	PROC longwelds()
		MoveJ [[-537.74,1528.93,225.26],[0.133056,-0.223334,0.96556,0.0105691],[1,-1,1,0],[9E+09,9E+09,9E+09,9E+09,9E+09,9E+09]], v1000, z50, tWeldGun;
		MoveJ [[-534.17,1676.79,-7.31],[0.13306,-0.223351,0.965556,0.0105536],[1,-1,1,0],[9E+09,9E+09,9E+09,9E+09,9E+09,9E+09]], v1000, z50, tWeldGun;
		ArcLStart [[-534.18,1676.79,-10.95],[0.13306,-0.223361,0.965554,0.0105477],[1,-1,1,0],[9E+09,9E+09,9E+09,9E+09,9E+09,9E+09]], v30, seam13, weld13, fine, tWeldGun;
		ArcL [[-544.58,1676.80,-10.94],[0.133063,-0.223367,0.965552,0.0105509],[1,-1,1,0],[9E+09,9E+09,9E+09,9E+09,9E+09,9E+09]], v30, seam13, weld13, z10, tWeldGun;
		ArcL [[-560.58,1676.80,-10.94],[0.133064,-0.223373,0.96555,0.0105523],[1,-1,1,0],[9E+09,9E+09,9E+09,9E+09,9E+09,9E+09]], v30, seam13, weld13, z10, tWeldGun;
		ArcLEnd [[-573.39,1676.78,-10.94],[0.133047,-0.223358,0.965556,0.0105449],[1,-1,1,0],[9E+09,9E+09,9E+09,9E+09,9E+09,9E+09]], v30, seam13, weld13, fine, tWeldGun;
		MoveL [[-573.40,1676.83,-5.98],[0.133038,-0.223382,0.965552,0.0105696],[1,-1,1,0],[9E+09,9E+09,9E+09,9E+09,9E+09,9E+09]], v50, z1, tWeldGun;
		MoveL [[-575.35,1723.62,-6.01],[0.133042,-0.223378,0.965552,0.0105594],[1,-1,1,0],[9E+09,9E+09,9E+09,9E+09,9E+09,9E+09]], v50, z1, tWeldGun;
		ArcLStart [[-575.34,1723.62,-15.03],[0.133047,-0.22338,0.965551,0.0105632],[1,-1,1,0],[9E+09,9E+09,9E+09,9E+09,9E+09,9E+09]], v30, seam13, weld13, fine, tWeldGun;
		ArcL [[-575.34,1697.62,-15.03],[0.133047,-0.22338,0.965551,0.0105669],[1,-1,1,0],[9E+09,9E+09,9E+09,9E+09,9E+09,9E+09]], v30, seam13, weld13, fine, tWeldGun;
		ArcL [[-575.35,1676.62,-15.02],[0.133043,-0.223381,0.965552,0.0105654],[1,-1,1,0],[9E+09,9E+09,9E+09,9E+09,9E+09,9E+09]], v30, seam13, weld13, fine, tWeldGun;
		ArcL [[-575.35,1655.62,-15.02],[0.13304,-0.223383,0.965551,0.010569],[1,-1,1,0],[9E+09,9E+09,9E+09,9E+09,9E+09,9E+09]], v30, seam13, weld13, fine, tWeldGun;
		ArcL [[-575.35,1632.62,-15.03],[0.133037,-0.22338,0.965553,0.0105659],[1,-1,1,0],[9E+09,9E+09,9E+09,9E+09,9E+09,9E+09]], v30, seam13, weld13, fine, tWeldGun;
		ArcLEnd [[-575.35,1606.61,-15.03],[0.133037,-0.223381,0.965552,0.0105613],[1,-1,1,0],[9E+09,9E+09,9E+09,9E+09,9E+09,9E+09]], v30, seam13, weld13, fine, tWeldGun;
		MoveL [[-575.35,1606.60,-1.09],[0.13303,-0.223389,0.965551,0.0105647],[1,-1,1,0],[9E+09,9E+09,9E+09,9E+09,9E+09,9E+09]], v50, z1, tWeldGun;
		MoveL [[-575.34,1585.59,-1.13],[0.133025,-0.223396,0.965551,0.0105485],[1,-1,1,0],[9E+09,9E+09,9E+09,9E+09,9E+09,9E+09]], v50, z1, tWeldGun;
		ArcLStart [[-574.36,1584.60,-16.12],[0.133023,-0.223401,0.96555,0.010553],[1,-1,1,0],[9E+09,9E+09,9E+09,9E+09,9E+09,9E+09]], v30, seam13, weld13\Weave:=weave1, fine, tWeldGun;
		ArcL [[-574.36,1575.59,-16.13],[0.13302,-0.2234,0.96555,0.0105496],[1,-1,1,0],[9E+09,9E+09,9E+09,9E+09,9E+09,9E+09]], v30, seam13, weld13\Weave:=weave1, fine, tWeldGun;
		ArcL [[-573.36,1542.60,-16.12],[0.133024,-0.223405,0.965549,0.0105554],[1,-1,1,0],[9E+09,9E+09,9E+09,9E+09,9E+09,9E+09]], v30, seam13, weld13\Weave:=weave1, fine, tWeldGun;
		ArcL [[-573.37,1523.59,-16.12],[0.133018,-0.223399,0.965551,0.010556],[1,-1,1,0],[9E+09,9E+09,9E+09,9E+09,9E+09,9E+09]], v30, seam13, weld13\Weave:=weave1, fine, tWeldGun;
		ArcLEnd [[-573.36,1500.60,-16.12],[0.133023,-0.223402,0.965549,0.0105616],[1,-1,1,0],[9E+09,9E+09,9E+09,9E+09,9E+09,9E+09]], v30, seam13, weld13\Weave:=weave1, fine, tWeldGun;
		MoveL [[-573.39,1500.62,-2.23],[0.132981,-0.22343,0.965549,0.0105695],[1,-1,1,0],[9E+09,9E+09,9E+09,9E+09,9E+09,9E+09]], v50, z1, tWeldGun;
		MoveL [[-573.39,1485.63,-2.25],[0.132987,-0.223446,0.965544,0.0105683],[1,-1,1,0],[9E+09,9E+09,9E+09,9E+09,9E+09,9E+09]], v50, z1, tWeldGun;
		ArcLStart [[-573.39,1485.63,-15.25],[0.132986,-0.223448,0.965544,0.0105658],[1,-1,1,0],[9E+09,9E+09,9E+09,9E+09,9E+09,9E+09]], v30, seam13, weld13\Weave:=weave1, fine, tWeldGun;
		ArcL [[-573.40,1464.62,-15.25],[0.132977,-0.223444,0.965546,0.0105643],[1,-1,1,0],[9E+09,9E+09,9E+09,9E+09,9E+09,9E+09]], v30, seam13, weld13\Weave:=weave1, fine, tWeldGun;
		ArcL [[-574.40,1445.63,-15.24],[0.132983,-0.223455,0.965542,0.0105677],[1,-1,1,0],[9E+09,9E+09,9E+09,9E+09,9E+09,9E+09]], v30, seam13, weld13\Weave:=weave1, fine, tWeldGun;
		ArcL [[-574.40,1425.64,-15.24],[0.132985,-0.223457,0.965542,0.0105723],[1,-1,1,0],[9E+09,9E+09,9E+09,9E+09,9E+09,9E+09]], v30, seam13, weld13\Weave:=weave1, fine, tWeldGun;
		ArcL [[-574.40,1404.65,-15.23],[0.132998,-0.223476,0.965536,0.0105691],[1,-1,1,0],[9E+09,9E+09,9E+09,9E+09,9E+09,9E+09]], v30, seam13, weld13\Weave:=weave1, fine, tWeldGun;
		ArcL [[-574.41,1387.63,-15.25],[0.132976,-0.223459,0.965543,0.0105667],[1,-1,1,0],[9E+09,9E+09,9E+09,9E+09,9E+09,9E+09]], v30, seam13, weld13\Weave:=weave1, fine, tWeldGun;
		ArcL [[-574.41,1369.63,-15.25],[0.132976,-0.22346,0.965542,0.0105621],[1,-1,1,0],[9E+09,9E+09,9E+09,9E+09,9E+09,9E+09]], v30, seam13, weld13\Weave:=weave1, fine, tWeldGun;
		ArcL [[-574.42,1347.62,-15.25],[0.132967,-0.223444,0.965547,0.0105695],[1,-1,1,0],[9E+09,9E+09,9E+09,9E+09,9E+09,9E+09]], v30, seam13, weld13\Weave:=weave1, fine, tWeldGun;
		ArcL [[-574.42,1329.62,-15.25],[0.132967,-0.223451,0.965546,0.0105668],[1,-1,1,0],[9E+09,9E+09,9E+09,9E+09,9E+09,9E+09]], v30, seam13, weld13\Weave:=weave1, fine, tWeldGun;
		ArcLEnd [[-575.42,1299.63,-13.24],[0.132972,-0.22346,0.965543,0.0105669],[1,-1,1,0],[9E+09,9E+09,9E+09,9E+09,9E+09,9E+09]], v30, seam13, weld13\Weave:=weave1, fine, tWeldGun;
		MoveL [[-575.42,1299.62,3.76],[0.132974,-0.223461,0.965542,0.0105603],[1,-1,1,0],[9E+09,9E+09,9E+09,9E+09,9E+09,9E+09]], v50, z1, tWeldGun;
		MoveL [[-575.41,1292.59,3.73],[0.13296,-0.223451,0.965547,0.0105324],[1,-1,1,0],[9E+09,9E+09,9E+09,9E+09,9E+09,9E+09]], v50, z1, tWeldGun;
		ArcLStart [[-576.42,1292.61,-13.26],[0.132961,-0.223463,0.965544,0.0105395],[1,-1,1,0],[9E+09,9E+09,9E+09,9E+09,9E+09,9E+09]], v30, seam13, weld13\Weave:=weave1, fine, tWeldGun;
		ArcLEnd [[-576.42,1112.60,-13.27],[0.132955,-0.223454,0.965547,0.010535],[1,-1,1,0],[9E+09,9E+09,9E+09,9E+09,9E+09,9E+09]], v30, seam13, weld13\Weave:=weave1, fine, tWeldGun;
		MoveL [[-576.42,1112.59,8.73],[0.132953,-0.22345,0.965548,0.0105277],[1,-1,1,0],[9E+09,9E+09,9E+09,9E+09,9E+09,9E+09]], v30, z1, tWeldGun;
		!MoveL [[-566.80,1587.36,103.77],[0.148014,0.588799,-0.740551,-0.288083],[1,-2,2,0],[9E+09,9E+09,9E+09,9E+09,9E+09,9E+09]], v30, z1, tWeldGun;
		!MoveL [[-566.80,1587.36,103.77],[0.148015,0.588798,-0.740552,-0.288083],[1,-2,2,0],[9E+09,9E+09,9E+09,9E+09,9E+09,9E+09]], v30, z1, tWeldGun;
		MoveJ [[-551.33,863.77,510.66],[0.15147,0.30253,-0.907678,-0.248302],[1,-1,1,0],[9E+09,9E+09,9E+09,9E+09,9E+09,9E+09]], vmax, z1, tWeldGun;
		MoveJ [[-551.34,773.91,9.99],[0.257685,0.331587,-0.885768,-0.197646],[1,-2,2,0],[9E+09,9E+09,9E+09,9E+09,9E+09,9E+09]], vmax, z1, tWeldGun;
		MoveL [[-569.03,771.59,1.41],[0.257705,0.331593,-0.885761,-0.197643],[1,-2,2,0],[9E+09,9E+09,9E+09,9E+09,9E+09,9E+09]], vmax, z1, tWeldGun;
		ArcLStart [[-569.03,771.58,-13.78],[0.257704,0.331613,-0.885754,-0.197643],[1,-2,2,0],[9E+09,9E+09,9E+09,9E+09,9E+09,9E+09]], v50, seam13, weld13\Weave:=weave1, fine, tWeldGun;
		ArcLEnd [[-568.49,798.58,-13.77],[0.257712,0.331608,-0.885753,-0.197645],[1,-2,2,0],[9E+09,9E+09,9E+09,9E+09,9E+09,9E+09]], v50, seam13, weld13\Weave:=weave1, fine, tWeldGun;
		MoveL [[-568.49,798.57,-7.98],[0.257716,0.331598,-0.885756,-0.197639],[1,-2,2,0],[9E+09,9E+09,9E+09,9E+09,9E+09,9E+09]], vmax, z1, tWeldGun;
		MoveL [[-567.50,823.73,-8.00],[0.257718,0.33163,-0.885749,-0.197615],[1,-2,2,0],[9E+09,9E+09,9E+09,9E+09,9E+09,9E+09]], vmax, z1, tWeldGun;
		ArcLStart [[-569.72,823.72,-13.19],[0.25773,0.331648,-0.88574,-0.197612],[1,-2,2,0],[9E+09,9E+09,9E+09,9E+09,9E+09,9E+09]], v50, seam13, weld13\Weave:=weave1, fine, tWeldGun;
		ArcLEnd [[-568.63,850.44,-13.40],[0.257728,0.331633,-0.885747,-0.197607],[1,-2,2,0],[9E+09,9E+09,9E+09,9E+09,9E+09,9E+09]], v50, seam13, weld13\Weave:=weave1, fine, tWeldGun;
		MoveL [[-568.64,850.44,-6.99],[0.257739,0.331614,-0.88575,-0.197611],[1,-2,2,0],[9E+09,9E+09,9E+09,9E+09,9E+09,9E+09]], vmax, z1, tWeldGun;
		MoveL [[-567.78,877.79,-7.01],[0.257734,0.331631,-0.885748,-0.1976],[1,-2,2,0],[9E+09,9E+09,9E+09,9E+09,9E+09,9E+09]], vmax, z1, tWeldGun;
		ArcLStart [[-568.78,876.58,-13.99],[0.257742,0.331637,-0.885742,-0.197602],[1,-2,2,0],[9E+09,9E+09,9E+09,9E+09,9E+09,9E+09]], v40, seam13, weld13\Weave:=weave1, fine, tWeldGun;
		ArcLEnd [[-569.59,895.98,-14.18],[0.257742,0.331687,-0.885727,-0.197589],[1,-2,2,0],[9E+09,9E+09,9E+09,9E+09,9E+09,9E+09]], v40, seam13, weld13\Weave:=weave1, fine, tWeldGun;
		MoveL [[-569.52,896.01,-8.19],[0.257699,0.331627,-0.885753,-0.197628],[1,-2,2,0],[9E+09,9E+09,9E+09,9E+09,9E+09,9E+09]], vmax, z1, tWeldGun;
		MoveL [[-569.26,927.41,-8.18],[0.257701,0.331632,-0.885751,-0.197629],[1,-2,2,0],[9E+09,9E+09,9E+09,9E+09,9E+09,9E+09]], vmax, z1, tWeldGun;
		ArcLStart [[-569.27,927.40,-14.18],[0.257703,0.331665,-0.88574,-0.197617],[1,-2,2,0],[9E+09,9E+09,9E+09,9E+09,9E+09,9E+09]], v40, seam13, weld13\Weave:=weave1, fine, tWeldGun;
		ArcLEnd [[-569.21,949.78,-14.59],[0.25771,0.331643,-0.885747,-0.197614],[1,-2,2,0],[9E+09,9E+09,9E+09,9E+09,9E+09,9E+09]], v40, seam13, weld13\Weave:=weave1, fine, tWeldGun;
		MoveL [[-569.21,949.78,-8.79],[0.257712,0.331634,-0.88575,-0.197614],[1,-2,2,0],[9E+09,9E+09,9E+09,9E+09,9E+09,9E+09]], vmax, z1, tWeldGun;
		MoveL [[-569.11,978.39,-8.78],[0.257713,0.331647,-0.885744,-0.197616],[1,-2,2,0],[9E+09,9E+09,9E+09,9E+09,9E+09,9E+09]], vmax, z1, tWeldGun;
		ArcLStart [[-569.11,978.38,-14.98],[0.257714,0.331662,-0.885739,-0.197612],[1,-2,2,0],[9E+09,9E+09,9E+09,9E+09,9E+09,9E+09]], v30, seam13, weld13\Weave:=weave1, fine, tWeldGun;
		ArcLEnd [[-569.11,1004.99,-14.97],[0.257723,0.331638,-0.885744,-0.197621],[1,-2,2,0],[9E+09,9E+09,9E+09,9E+09,9E+09,9E+09]], v30, seam13, weld13\Weave:=weave1, fine, tWeldGun;
		MoveL [[-569.11,1004.98,-9.57],[0.257725,0.331632,-0.885746,-0.197618],[1,-2,2,0],[9E+09,9E+09,9E+09,9E+09,9E+09,9E+09]], vmax, z1, tWeldGun;
		MoveL [[-568.66,1030.78,-9.56],[0.257723,0.331657,-0.885737,-0.197616],[1,-2,2,0],[9E+09,9E+09,9E+09,9E+09,9E+09,9E+09]], vmax, z1, tWeldGun;
		ArcLStart [[-569.26,1030.55,-15.38],[0.257732,0.331656,-0.885738,-0.197603],[1,-2,2,0],[9E+09,9E+09,9E+09,9E+09,9E+09,9E+09]], v30, seam13, weld13\Weave:=weave1, fine, tWeldGun;
		ArcLEnd [[-568.86,1056.55,-15.38],[0.257739,0.331642,-0.885741,-0.197603],[1,-2,2,0],[9E+09,9E+09,9E+09,9E+09,9E+09,9E+09]], v30, seam13, weld13\Weave:=weave1, fine, tWeldGun;
		MoveL [[-568.86,1056.55,-6.38],[0.257746,0.331635,-0.885742,-0.197603],[1,-2,2,0],[9E+09,9E+09,9E+09,9E+09,9E+09,9E+09]], vmax, z1, tWeldGun;
		MoveL [[-567.90,1082.34,-6.38],[0.257746,0.331649,-0.885737,-0.197601],[1,-2,2,0],[9E+09,9E+09,9E+09,9E+09,9E+09,9E+09]], vmax, z1, tWeldGun;
		ArcLStart [[-568.70,1082.12,-15.98],[0.257751,0.33165,-0.885737,-0.197592],[1,-2,2,0],[9E+09,9E+09,9E+09,9E+09,9E+09,9E+09]], v20, seam13, weld13\Weave:=weave1, fine, tWeldGun;
		ArcLEnd [[-568.24,1107.52,-15.98],[0.257752,0.331667,-0.885731,-0.19759],[1,-2,2,0],[9E+09,9E+09,9E+09,9E+09,9E+09,9E+09]], v20, seam13, weld13\Weave:=weave1, fine, tWeldGun;
		MoveL [[-568.24,1107.51,-8.98],[0.257762,0.331649,-0.885734,-0.197593],[1,-2,2,0],[9E+09,9E+09,9E+09,9E+09,9E+09,9E+09]], vmax, z1, tWeldGun;
		MoveL [[-568.24,1133.52,-8.97],[0.257758,0.331653,-0.885733,-0.197595],[1,-2,2,0],[9E+09,9E+09,9E+09,9E+09,9E+09,9E+09]], vmax, z1, tWeldGun;
		ArcLStart [[-568.25,1133.51,-15.58],[0.257762,0.331659,-0.885732,-0.197589],[1,-2,2,0],[9E+09,9E+09,9E+09,9E+09,9E+09,9E+09]], v20, seam13, weld13\Weave:=weave1, fine, tWeldGun;
		ArcLEnd [[-568.25,1158.71,-15.60],[0.257768,0.331651,-0.885734,-0.197582],[1,-2,2,0],[9E+09,9E+09,9E+09,9E+09,9E+09,9E+09]], v20, seam13, weld13\Weave:=weave1, fine, tWeldGun;
		MoveL [[-568.24,1158.69,-5.60],[0.257781,0.331624,-0.885741,-0.197583],[1,-2,2,0],[9E+09,9E+09,9E+09,9E+09,9E+09,9E+09]], vmax, z1, tWeldGun;
		MoveL [[-567.89,1183.28,-5.61],[0.257781,0.331645,-0.885735,-0.197572],[1,-2,2,0],[9E+09,9E+09,9E+09,9E+09,9E+09,9E+09]], vmax, z1, tWeldGun;
		ArcLStart [[-568.69,1183.27,-16.02],[0.257789,0.331641,-0.885736,-0.197564],[1,-2,2,0],[9E+09,9E+09,9E+09,9E+09,9E+09,9E+09]], v10, seam13, weld13\Weave:=weave1, fine, tWeldGun;
		ArcLEnd [[-568.49,1207.45,-16.03],[0.257793,0.331641,-0.885736,-0.197559],[1,-2,2,0],[9E+09,9E+09,9E+09,9E+09,9E+09,9E+09]], v10, seam13, weld13\Weave:=weave1, fine, tWeldGun;
		MoveL [[-568.49,1207.45,-8.63],[0.257801,0.331631,-0.885737,-0.197558],[1,-2,2,0],[9E+09,9E+09,9E+09,9E+09,9E+09,9E+09]], vmax, z1, tWeldGun;
		MoveL [[-568.50,1234.87,-8.62],[0.257795,0.331647,-0.885732,-0.197564],[1,-2,2,0],[9E+09,9E+09,9E+09,9E+09,9E+09,9E+09]], vmax, z1, tWeldGun;
		ArcLStart [[-568.49,1234.85,-16.22],[0.25779,0.331666,-0.885728,-0.197556],[1,-2,2,0],[9E+09,9E+09,9E+09,9E+09,9E+09,9E+09]], v10, seam13, weld13\Weave:=weave1, fine, tWeldGun;
		ArcLEnd [[-568.03,1261.25,-16.22],[0.257799,0.331652,-0.88573,-0.19756],[1,-2,2,0],[9E+09,9E+09,9E+09,9E+09,9E+09,9E+09]], v10, seam13, weld13\Weave:=weave1, fine, tWeldGun;
		MoveL [[-568.04,1261.25,-8.21],[0.257811,0.331635,-0.885732,-0.197564],[1,-2,2,0],[9E+09,9E+09,9E+09,9E+09,9E+09,9E+09]], vmax, z1, tWeldGun;
		MoveL [[-567.52,1287.24,-8.21],[0.257803,0.331653,-0.885727,-0.197564],[1,-2,2,0],[9E+09,9E+09,9E+09,9E+09,9E+09,9E+09]], vmax, z1, tWeldGun;
		ArcLStart [[-568.52,1287.23,-15.81],[0.257806,0.331656,-0.885726,-0.197561],[1,-2,2,0],[9E+09,9E+09,9E+09,9E+09,9E+09,9E+09]], v60, seam13, weld13\Weave:=weave1, fine, tWeldGun;
		ArcLEnd [[-568.38,1312.23,-16.00],[0.257804,0.331674,-0.88572,-0.197561],[1,-2,2,0],[9E+09,9E+09,9E+09,9E+09,9E+09,9E+09]], v60, seam13, weld13\Weave:=weave1, fine, tWeldGun;
		MoveL [[-568.37,1312.22,-9.20],[0.257819,0.33164,-0.885728,-0.197564],[1,-2,2,0],[9E+09,9E+09,9E+09,9E+09,9E+09,9E+09]], vmax, z1, tWeldGun;
		MoveL [[-566.34,1338.40,-9.21],[0.257813,0.331671,-0.885721,-0.19755],[1,-2,2,0],[9E+09,9E+09,9E+09,9E+09,9E+09,9E+09]], vmax, z1, tWeldGun;
		ArcLStart [[-567.35,1338.00,-18.39],[0.257823,0.331668,-0.885717,-0.197557],[1,-2,2,0],[9E+09,9E+09,9E+09,9E+09,9E+09,9E+09]], v60, seam13, weld13\Weave:=weave1, fine, tWeldGun;
		ArcLEnd [[-566.97,1362.99,-18.40],[0.257825,0.331676,-0.885715,-0.197551],[1,-2,2,0],[9E+09,9E+09,9E+09,9E+09,9E+09,9E+09]], v60, seam13, weld13\Weave:=weave1, fine, tWeldGun;
		!WorldAccLim\Off;
		MoveL [[-566.97,1362.98,-3.40],[0.257832,0.33166,-0.885719,-0.197554],[1,-2,2,0],[9E+09,9E+09,9E+09,9E+09,9E+09,9E+09]], vmax, z1, tWeldGun;
		MoveJ [[-569.01,1526.90,-0.76],[0.343671,0.343727,-0.853199,-0.189191],[1,-2,2,0],[9E+09,9E+09,9E+09,9E+09,9E+09,9E+09]], vmax, z1, tWeldGun;
		ArcLStart [[-570.01,1526.88,-19.38],[0.343676,0.343732,-0.853197,-0.189182],[1,-2,2,0],[9E+09,9E+09,9E+09,9E+09,9E+09,9E+09]], v30, seam13, weld13\Weave:=weave1, fine, tWeldGun;
		ArcLEnd [[-569.62,1552.28,-19.38],[0.343683,0.343722,-0.853198,-0.189184],[1,-2,2,0],[9E+09,9E+09,9E+09,9E+09,9E+09,9E+09]], v30, seam13, weld13\Weave:=weave1, fine, tWeldGun;
		MoveL [[-569.62,1552.28,-11.37],[0.343694,0.343705,-0.853199,-0.189192],[1,-2,2,0],[9E+09,9E+09,9E+09,9E+09,9E+09,9E+09]], vmax, z1, tWeldGun;
		MoveL [[-569.12,1581.67,-11.38],[0.343681,0.343726,-0.853198,-0.189184],[1,-2,1,0],[9E+09,9E+09,9E+09,9E+09,9E+09,9E+09]], vmax, z1, tWeldGun;
		ArcLStart [[-569.12,1581.67,-19.57],[0.343687,0.343722,-0.853196,-0.189187],[1,-2,2,0],[9E+09,9E+09,9E+09,9E+09,9E+09,9E+09]], v30, seam13, weld13\Weave:=weave1, fine, tWeldGun;
		ArcLEnd [[-568.85,1605.87,-19.56],[0.343691,0.34372,-0.853194,-0.189191],[1,-2,1,0],[9E+09,9E+09,9E+09,9E+09,9E+09,9E+09]], v30, seam13, weld13\Weave:=weave1, fine, tWeldGun;
		MoveL [[-568.85,1605.87,-2.98],[0.343682,0.343726,-0.853196,-0.189187],[1,-1,1,0],[9E+09,9E+09,9E+09,9E+09,9E+09,9E+09]], vmax, z1, tWeldGun;
		MoveL [[-568.53,1630.66,-3.00],[0.343686,0.34372,-0.853198,-0.189182],[1,1,-1,1],[9E+09,9E+09,9E+09,9E+09,9E+09,9E+09]], vmax, z1, tWeldGun;
		ArcLStart [[-570.74,1630.45,-19.81],[0.343708,0.343698,-0.853198,-0.189185],[1,1,-1,1],[9E+09,9E+09,9E+09,9E+09,9E+09,9E+09]], v30, seam13, weld13\Weave:=weave1, fine, tWeldGun;
		ArcLEnd [[-571.08,1657.04,-19.81],[0.343713,0.343698,-0.853195,-0.189186],[1,1,-1,1],[9E+09,9E+09,9E+09,9E+09,9E+09,9E+09]], v30, seam13, weld13\Weave:=weave1, fine, tWeldGun;
		MoveL [[-571.08,1657.05,-10.39],[0.343723,0.343675,-0.853198,-0.189199],[1,1,-1,1],[9E+09,9E+09,9E+09,9E+09,9E+09,9E+09]], vmax, z1, tWeldGun;
		MoveL [[-569.60,1683.62,-10.40],[0.343722,0.343687,-0.853195,-0.189194],[1,1,-1,1],[9E+09,9E+09,9E+09,9E+09,9E+09,9E+09]], vmax, z1, tWeldGun;
		ArcLStart [[-570.40,1683.62,-19.59],[0.343729,0.343674,-0.853196,-0.1892],[1,1,-1,1],[9E+09,9E+09,9E+09,9E+09,9E+09,9E+09]], v30, seam13, weld13\Weave:=weave1, fine, tWeldGun;
		ArcLEnd [[-569.44,1706.01,-19.59],[0.343736,0.343668,-0.853195,-0.1892],[1,1,-1,1],[9E+09,9E+09,9E+09,9E+09,9E+09,9E+09]], v30, seam13, weld13\Weave:=weave1, fine, tWeldGun;
		MoveL [[-569.44,1706.01,-12.58],[0.343736,0.343663,-0.853196,-0.189202],[1,1,-1,1],[9E+09,9E+09,9E+09,9E+09,9E+09,9E+09]], vmax, z1, tWeldGun;
		MoveL [[-568.95,1728.80,-12.59],[0.343738,0.343665,-0.853195,-0.189201],[1,1,-1,1],[9E+09,9E+09,9E+09,9E+09,9E+09,9E+09]], vmax, z1, tWeldGun;
		ArcLStart [[-568.57,1727.28,-19.96],[0.343763,0.34365,-0.853188,-0.189216],[1,1,-1,1],[9E+09,9E+09,9E+09,9E+09,9E+09,9E+09]], v30, seam13, weld13\Weave:=weave1, fine, tWeldGun;
		ArcLEnd [[-568.38,1754.27,-19.94],[0.343779,0.343637,-0.853184,-0.189226],[1,1,-1,1],[9E+09,9E+09,9E+09,9E+09,9E+09,9E+09]], v30, seam13, weld13\Weave:=weave1, fine, tWeldGun;
		MoveL [[-568.37,1754.26,-12.54],[0.343778,0.343636,-0.853186,-0.189221],[1,1,-1,1],[9E+09,9E+09,9E+09,9E+09,9E+09,9E+09]], vmax, z1, tWeldGun;
		MoveL [[-568.19,1780.66,-12.54],[0.343782,0.343632,-0.853186,-0.189224],[1,1,-1,1],[9E+09,9E+09,9E+09,9E+09,9E+09,9E+09]], vmax, z1, tWeldGun;
		ArcLStart [[-568.19,1779.25,-19.93],[0.343783,0.343638,-0.853184,-0.18922],[1,1,-1,1],[9E+09,9E+09,9E+09,9E+09,9E+09,9E+09]], v30, seam13, weld13\Weave:=weave1, fine, tWeldGun;
		ArcLEnd [[-567.11,1804.25,-19.92],[0.343792,0.343628,-0.853182,-0.189228],[1,1,-2,1],[9E+09,9E+09,9E+09,9E+09,9E+09,9E+09]], v30, seam13, weld13\Weave:=weave1, fine, tWeldGun;
		MoveL [[-567.12,1804.23,78.28],[0.343797,0.343622,-0.853184,-0.189223],[1,1,-2,1],[9E+09,9E+09,9E+09,9E+09,9E+09,9E+09]], vmax, z1, tWeldGun;
		ArcLStart [[-567.96,1824.13,-22.58],[0.321693,0.391445,-0.845647,-0.167826],[1,-1,0,0],[9E+09,9E+09,9E+09,9E+09,9E+09,9E+09]], v30, seam13, weld13\Weave:=weave1, fine, tWeldGun;
		ArcLEnd [[-567.85,1853.11,-22.61],[0.321723,0.391404,-0.845654,-0.16783],[1,-1,0,0],[9E+09,9E+09,9E+09,9E+09,9E+09,9E+09]], v30, seam13, weld13\Weave:=weave1, fine, tWeldGun;
		MoveL [[-567.86,1853.06,64.86],[0.321729,0.391441,-0.845624,-0.167883],[1,-1,0,0],[9E+09,9E+09,9E+09,9E+09,9E+09,9E+09]], v30, z1, tWeldGun;
		MoveL [[-589.56,1806.04,41.58],[0.316409,0.386415,-0.856917,-0.127529],[1,-1,0,0],[9E+09,9E+09,9E+09,9E+09,9E+09,9E+09]], v30, z1, tWeldGun;
		MoveL [[-565.44,1418.25,0.00],[0.316355,0.386506,-0.856899,-0.127503],[1,-1,1,0],[9E+09,9E+09,9E+09,9E+09,9E+09,9E+09]], v30, z1, tWeldGun;
		ArcLStart [[-566.84,1418.23,-21.63],[0.31636,0.386522,-0.856891,-0.127501],[1,-1,1,0],[9E+09,9E+09,9E+09,9E+09,9E+09,9E+09]], v30, seam13, weld13\Weave:=weave1, fine, tWeldGun;
		ArcLEnd [[-566.32,1443.02,-21.63],[0.316365,0.386514,-0.856892,-0.127502],[1,-1,1,0],[9E+09,9E+09,9E+09,9E+09,9E+09,9E+09]], v30, seam13, weld13\Weave:=weave1, fine, tWeldGun;
		MoveL [[-566.32,1443.03,10.49],[0.316366,0.386508,-0.856894,-0.127504],[1,-1,1,0],[9E+09,9E+09,9E+09,9E+09,9E+09,9E+09]], v30, z1, tWeldGun;
		MoveL [[-565.57,1462.70,10.49],[0.316366,0.386516,-0.85689,-0.127504],[1,-1,1,0],[9E+09,9E+09,9E+09,9E+09,9E+09,9E+09]], v30, z1, tWeldGun;
		ArcLStart [[-565.57,1456.12,-20.37],[0.316374,0.386523,-0.856885,-0.127501],[1,-1,1,0],[9E+09,9E+09,9E+09,9E+09,9E+09,9E+09]], v30, seam13, weld13\Weave:=weave1, fine, tWeldGun;
		ArcLEnd [[-565.36,1487.97,-20.36],[0.316378,0.386527,-0.856881,-0.127502],[1,-1,1,0],[9E+09,9E+09,9E+09,9E+09,9E+09,9E+09]], v30, seam13, weld13\Weave:=weave1, fine, tWeldGun;
		MoveL [[-565.36,1487.97,2.46],[0.31638,0.386514,-0.856886,-0.127504],[1,-1,1,0],[9E+09,9E+09,9E+09,9E+09,9E+09,9E+09]], v30, z1, tWeldGun;
		MoveL [[-559.76,1655.50,2.46],[0.316384,0.386516,-0.856884,-0.127503],[1,-1,0,0],[9E+09,9E+09,9E+09,9E+09,9E+09,9E+09]], vmax, z1, tWeldGun;
		ArcLStart [[-565.96,1655.48,-22.55],[0.316397,0.386513,-0.856881,-0.127497],[1,-1,1,0],[9E+09,9E+09,9E+09,9E+09,9E+09,9E+09]], v30, seam13, weld13\Weave:=weave1, fine, tWeldGun;
		ArcLEnd [[-566.37,1676.08,-22.53],[0.316408,0.386509,-0.856879,-0.127501],[1,-1,0,0],[9E+09,9E+09,9E+09,9E+09,9E+09,9E+09]], v30, seam13, weld13\Weave:=weave1, fine, tWeldGun;
		MoveL [[-566.36,1676.08,-13.72],[0.316407,0.386508,-0.85688,-0.1275],[1,-1,0,0],[9E+09,9E+09,9E+09,9E+09,9E+09,9E+09]], vmax, z1, tWeldGun;
		MoveL [[-565.20,1705.25,-13.73],[0.316413,0.386506,-0.856879,-0.127497],[1,-1,0,0],[9E+09,9E+09,9E+09,9E+09,9E+09,9E+09]], vmax, z1, tWeldGun;
		ArcLStart [[-565.20,1705.25,-23.32],[0.316413,0.386514,-0.856875,-0.1275],[1,-1,0,0],[9E+09,9E+09,9E+09,9E+09,9E+09,9E+09]], v30, seam13, weld13\Weave:=weave1, fine, tWeldGun;
		ArcLEnd [[-564.28,1720.82,-23.32],[0.316416,0.386511,-0.856874,-0.127501],[1,-1,0,0],[9E+09,9E+09,9E+09,9E+09,9E+09,9E+09]], v30, seam13, weld13\Weave:=weave1, fine, tWeldGun;
		MoveL [[-564.28,1720.81,-13.32],[0.316421,0.3865,-0.856878,-0.1275],[1,-1,0,0],[9E+09,9E+09,9E+09,9E+09,9E+09,9E+09]], vmax, z1, tWeldGun;
		MoveL [[-562.15,1754.27,-13.31],[0.316419,0.386514,-0.856873,-0.127498],[1,-1,0,0],[9E+09,9E+09,9E+09,9E+09,9E+09,9E+09]], vmax, z1, tWeldGun;
		ArcLStart [[-564.55,1753.27,-22.70],[0.316421,0.386527,-0.856865,-0.127503],[1,-1,0,0],[9E+09,9E+09,9E+09,9E+09,9E+09,9E+09]], v30, seam13, weld13\Weave:=weave1, fine, tWeldGun;
		ArcLEnd [[-564.27,1773.06,-22.70],[0.316431,0.386515,-0.856867,-0.127504],[1,-1,0,0],[9E+09,9E+09,9E+09,9E+09,9E+09,9E+09]], v30, seam13, weld13\Weave:=weave1, fine, tWeldGun;
		MoveL [[-564.27,1773.06,-14.70],[0.316433,0.38651,-0.856868,-0.127506],[1,-1,0,0],[9E+09,9E+09,9E+09,9E+09,9E+09,9E+09]], vmax, z1, tWeldGun;
		MoveL [[-562.44,1801.51,-11.84],[0.301948,0.358368,-0.858842,-0.20686],[1,-1,1,0],[9E+09,9E+09,9E+09,9E+09,9E+09,9E+09]], vmax, z1, tWeldGun;
		ArcLStart [[-562.45,1801.50,-21.64],[0.301956,0.358366,-0.858839,-0.206864],[1,-1,1,0],[9E+09,9E+09,9E+09,9E+09,9E+09,9E+09]], v30, seam13, weld13\Weave:=weave1, fine, tWeldGun;
		ArcLEnd [[-561.95,1822.85,-21.66],[0.301963,0.358358,-0.858841,-0.206859],[1,-1,1,0],[9E+09,9E+09,9E+09,9E+09,9E+09,9E+09]], v30, seam13, weld13\Weave:=weave1, fine, tWeldGun;
		MoveL [[-562.07,1822.86,13.32],[0.302053,0.358369,-0.858792,-0.20691],[1,-1,1,0],[9E+09,9E+09,9E+09,9E+09,9E+09,9E+09]], vmax, z1, tWeldGun;
	ENDPROC
	PROC rRUNSide1A200()
           	rTestPosTop;
		TPWrite "Side 1 A";
		MoveJ pSafeS1, vmax, fine, tWeldGun;
		!Code Goes Here
		MoveJ pSafeS181, vmax, fine, tWeldGun;
		SingArea\Wrist;
		MoveJ [[1181.97,1536.60,299.24],[0.0635588,0.517232,-0.779106,0.348462],[0,1,-3,1],[9E+09,9E+09,9E+09,9E+09,9E+09,9E+09]], vmax, z10, tWeldGun;
		MoveL [[1181.95,1536.61,-4.61],[0.0635699,0.51724,-0.779104,0.348453],[0,1,-2,1],[9E+09,9E+09,9E+09,9E+09,9E+09,9E+09]], v1000, z10, tWeldGun;
		ArcLStart [[1183.34,1532.14,-10.38],[0.0432656,0.526366,-0.780926,0.333501],[0,1,-2,1],[9E+09,9E+09,9E+09,9E+09,9E+09,9E+09]], v10, seam13, weld13\Weave:=weave1, fine, tWeldGun;
		ArcLEnd [[1206.22,1532.24,-10.36],[0.0432175,0.526382,-0.780937,0.333453],[0,1,-2,1],[9E+09,9E+09,9E+09,9E+09,9E+09,9E+09]], v10, seam13, weld13\Weave:=weave1, fine, tWeldGun;
		MoveL [[1204.62,1537.22,-4.87],[0.0635798,0.517232,-0.779109,0.348451],[0,1,-2,1],[9E+09,9E+09,9E+09,9E+09,9E+09,9E+09]], vmax, z10, tWeldGun;
		MoveL [[863.66,1538.85,77.89],[0.0635666,0.517243,-0.779097,0.348464],[0,1,-2,1],[9E+09,9E+09,9E+09,9E+09,9E+09,9E+09]], vmax, z10, tWeldGun;
		MoveJ [[861.58,1461.21,260.09],[0.14949,-0.376148,-0.839997,-0.361347],[0,1,-1,1],[9E+09,9E+09,9E+09,9E+09,9E+09,9E+09]], vmax, z10, tWeldGun;
		MoveL [[863.22,1468.67,-10.11],[0.149522,-0.376221,-0.839963,-0.361336],[0,1,-1,1],[9E+09,9E+09,9E+09,9E+09,9E+09,9E+09]], v1000, z10, tWeldGun;
		ArcLStart [[866.37,1476.97,-12.05],[0.0874714,-0.401117,-0.850564,-0.328626],[0,1,-1,1],[9E+09,9E+09,9E+09,9E+09,9E+09,9E+09]], v10, seam13, weld13\Weave:=weave1, fine, tWeldGun;
		ArcLEnd [[894.17,1477.17,-12.05],[0.0874956,-0.401178,-0.850524,-0.328648],[0,1,-1,1],[9E+09,9E+09,9E+09,9E+09,9E+09,9E+09]], v10, seam13, weld13\Weave:=weave1, fine, tWeldGun;
		MoveL [[886.08,1463.03,-7.28],[0.149478,-0.376156,-0.840008,-0.361317],[0,1,-1,1],[9E+09,9E+09,9E+09,9E+09,9E+09,9E+09]], vmax, z10, tWeldGun;
		MoveJ [[863.35,1506.96,224.59],[0.0635605,0.517248,-0.779091,0.348471],[0,1,-2,1],[9E+09,9E+09,9E+09,9E+09,9E+09,9E+09]], vmax, z10, tWeldGun;
		MoveL [[863.49,1538.37,-7.85],[0.0635592,0.51724,-0.779122,0.348415],[0,1,-2,1],[9E+09,9E+09,9E+09,9E+09,9E+09,9E+09]], vmax, z10, tWeldGun;
		ArcLStart [[863.39,1533.35,-9.29],[0.0457935,0.525049,-0.780128,0.337086],[0,1,-2,1],[9E+09,9E+09,9E+09,9E+09,9E+09,9E+09]], v10, seam13, weld13\Weave:=weave1, fine, tWeldGun;
		ArcLEnd [[889.04,1533.30,-8.67],[0.0457782,0.525087,-0.780065,0.337177],[0,1,-2,1],[9E+09,9E+09,9E+09,9E+09,9E+09,9E+09]], v10, seam13, weld13\Weave:=weave1, fine, tWeldGun;
		MoveL [[887.77,1539.90,182.89],[0.0635615,0.517251,-0.779088,0.348474],[0,1,-2,1],[9E+09,9E+09,9E+09,9E+09,9E+09,9E+09]], vmax, z10, tWeldGun;
		MoveJ [[1182.52,1470.34,61.27],[0.149538,-0.376243,-0.839941,-0.361358],[0,1,-1,1],[9E+09,9E+09,9E+09,9E+09,9E+09,9E+09]], vmax, z10, tWeldGun;
		MoveL [[1181.55,1464.42,-9.30],[0.148332,-0.500326,-0.790399,-0.320847],[0,1,-1,1],[9E+09,9E+09,9E+09,9E+09,9E+09,9E+09]], v1000, z10, tWeldGun;
		ArcLStart [[1177.33,1473.60,-12.87],[0.148345,-0.500351,-0.790382,-0.320842],[0,1,-1,1],[9E+09,9E+09,9E+09,9E+09,9E+09,9E+09]], v10, seam13, weld13\Weave:=weave1, fine, tWeldGun;
		ArcLEnd [[1207.54,1473.57,-12.86],[0.148337,-0.500345,-0.790386,-0.320845],[0,1,-1,1],[9E+09,9E+09,9E+09,9E+09,9E+09,9E+09]], v10, seam13, weld13\Weave:=weave1, fine, tWeldGun;
		MoveL [[1206.87,1462.04,-3.48],[0.148351,-0.500349,-0.790363,-0.320889],[0,1,-1,1],[9E+09,9E+09,9E+09,9E+09,9E+09,9E+09]], vmax, z10, tWeldGun;
		MoveL [[1203.94,921.98,77.52],[0.149416,-0.376356,-0.839957,-0.361252],[0,1,-1,1],[9E+09,9E+09,9E+09,9E+09,9E+09,9E+09]], vmax, z10, tWeldGun;
		MoveL [[1209.28,920.32,-0.95],[0.0811338,-0.402507,-0.844244,-0.344469],[0,1,-1,1],[9E+09,9E+09,9E+09,9E+09,9E+09,9E+09]], v1000, z10, tWeldGun;
		ArcLStart [[1208.91,928.66,-10.99],[0.081096,-0.402552,-0.84423,-0.344458],[0,1,-1,1],[9E+09,9E+09,9E+09,9E+09,9E+09,9E+09]], v10, seam13, weld13\Weave:=weave1, fine, tWeldGun;
		ArcLEnd [[1180.12,929.43,-11.01],[0.0811029,-0.402583,-0.844212,-0.344465],[0,1,0,1],[9E+09,9E+09,9E+09,9E+09,9E+09,9E+09]], v10, seam13, weld13\Weave:=weave1, fine, tWeldGun;
		MoveL [[1182.60,918.33,-2.85],[0.0811745,-0.402551,-0.844212,-0.344485],[0,1,0,1],[9E+09,9E+09,9E+09,9E+09,9E+09,9E+09]], vmax, z10, tWeldGun;
		MoveL [[883.71,921.14,-1.64],[0.149424,-0.37639,-0.839933,-0.361269],[0,1,0,1],[9E+09,9E+09,9E+09,9E+09,9E+09,9E+09]], vmax, z10, tWeldGun;
		MoveL [[891.05,920.87,-4.97],[0.15161,-0.376469,-0.855824,-0.320705],[0,1,-1,1],[9E+09,9E+09,9E+09,9E+09,9E+09,9E+09]], v1000, z10, tWeldGun;
		ArcLStart [[890.95,930.44,-12.87],[0.151512,-0.376481,-0.855837,-0.320703],[0,1,-1,1],[9E+09,9E+09,9E+09,9E+09,9E+09,9E+09]], v10, seam13, weld13\Weave:=weave1, fine, tWeldGun;
		ArcLEnd [[864.65,932.03,-12.68],[0.151535,-0.376589,-0.85577,-0.320744],[0,1,-1,1],[9E+09,9E+09,9E+09,9E+09,9E+09,9E+09]], v10, seam13, weld13\Weave:=weave1, fine, tWeldGun;
		MoveL [[866.54,921.07,-4.87],[0.151523,-0.376433,-0.855874,-0.320656],[0,1,-1,1],[9E+09,9E+09,9E+09,9E+09,9E+09,9E+09]], v100, z10, tWeldGun;
		MoveL [[861.26,919.79,117.88],[0.149443,-0.376442,-0.8399,-0.361285],[0,1,-1,1],[9E+09,9E+09,9E+09,9E+09,9E+09,9E+09]], vmax, z0, tWeldGun;
		MoveJ [[868.17,991.07,127.71],[0.0426372,-0.330552,0.858067,-0.39069],[0,1,-2,1],[9E+09,9E+09,9E+09,9E+09,9E+09,9E+09]], vmax, z0, tWeldGun;
		MoveL [[863.71,988.79,-2.92],[0.042941,-0.330682,0.857982,-0.390734],[0,0,-2,1],[9E+09,9E+09,9E+09,9E+09,9E+09,9E+09]], v1000, z10, tWeldGun;
		ArcLStart [[861.89,984.77,-9.70],[0.0429638,-0.330722,0.857953,-0.39076],[0,0,-2,1],[9E+09,9E+09,9E+09,9E+09,9E+09,9E+09]], v10, seam13, weld13\Weave:=weave1, fine, tWeldGun;
		ArcLEnd [[889.87,985.15,-9.73],[0.0429414,-0.330754,0.857925,-0.390798],[0,0,-2,1],[9E+09,9E+09,9E+09,9E+09,9E+09,9E+09]], v10, seam13, weld13\Weave:=weave1, fine, tWeldGun;
		MoveL [[889.59,992.71,-6.61],[0.0430178,-0.330607,0.858002,-0.390745],[0,0,-2,1],[9E+09,9E+09,9E+09,9E+09,9E+09,9E+09]], vmax, z10, tWeldGun;
		MoveL [[889.59,992.73,75.52],[0.0430306,-0.330621,0.857997,-0.390743],[0,1,-2,1],[9E+09,9E+09,9E+09,9E+09,9E+09,9E+09]], vmax, z10, tWeldGun;
		MoveL [[1177.66,992.72,75.52],[0.0430182,-0.33062,0.857997,-0.390745],[0,0,-2,1],[9E+09,9E+09,9E+09,9E+09,9E+09,9E+09]], vmax, z10, tWeldGun;
		MoveL [[1185.35,990.20,-3.61],[0.0429073,-0.330578,0.858028,-0.390724],[0,0,-2,1],[9E+09,9E+09,9E+09,9E+09,9E+09,9E+09]], v1000, z10, tWeldGun;
		ArcLStart [[1176.08,984.61,-10.65],[0.0451953,-0.325527,0.859941,-0.390503],[0,0,-2,1],[9E+09,9E+09,9E+09,9E+09,9E+09,9E+09]], v10, seam13, weld13\Weave:=weave1, fine, tWeldGun;
		ArcLEnd [[1210.47,984.70,-10.67],[0.0451959,-0.325517,0.859949,-0.390493],[0,0,-2,1],[9E+09,9E+09,9E+09,9E+09,9E+09,9E+09]], v10, seam13, weld13\Weave:=weave1, fine, tWeldGun;
		MoveL [[1207.94,989.04,-11.16],[0.0429397,-0.330625,0.858002,-0.39074],[0,0,-2,1],[9E+09,9E+09,9E+09,9E+09,9E+09,9E+09]], v1000, z10, tWeldGun;
		MoveL [[1207.95,989.04,392.36],[0.0429563,-0.330627,0.857995,-0.39075],[0,1,-2,1],[9E+09,9E+09,9E+09,9E+09,9E+09,9E+09]], vmax, z10, tWeldGun;
		MoveJ [[194.09,1536.38,108.42],[0.0907205,-0.623393,0.712906,0.308084],[0,-1,0,1],[9E+09,9E+09,9E+09,9E+09,9E+09,9E+09]], vmax, z10, tWeldGun;
		MoveL [[194.09,1534.55,21.51],[0.0907097,-0.623392,0.712903,0.308096],[0,-1,0,1],[9E+09,9E+09,9E+09,9E+09,9E+09,9E+09]], vmax, z10, tWeldGun;
		ArcLStart [[190.35,1535.97,0.59],[0.0903662,-0.623335,0.713039,0.307999],[0,-1,0,1],[9E+09,9E+09,9E+09,9E+09,9E+09,9E+09]], v20, seam13, weld13\Weave:=weave1, fine, tWeldGun;
		ArcLEnd [[159.94,1535.93,0.55],[0.090343,-0.623341,0.713041,0.307988],[0,-1,0,1],[9E+09,9E+09,9E+09,9E+09,9E+09,9E+09]], v20, seam13, weld13\Weave:=weave1, fine, tWeldGun;
		MoveL [[158.09,1532.35,8.43],[0.0907075,-0.623402,0.712898,0.30809],[0,-1,0,1],[9E+09,9E+09,9E+09,9E+09,9E+09,9E+09]], vmax, z10, tWeldGun;
		MoveL [[-128.01,1535.58,7.69],[0.090663,-0.623378,0.712945,0.308043],[1,0,0,1],[9E+09,9E+09,9E+09,9E+09,9E+09,9E+09]], vmax, z10, tWeldGun;
		ArcLStart [[-127.83,1537.58,1.69],[0.0906477,-0.623383,0.712936,0.308058],[1,0,0,1],[9E+09,9E+09,9E+09,9E+09,9E+09,9E+09]], v20, seam13, weld13\Weave:=weave1, fine, tWeldGun;
		ArcLEnd [[-158.66,1537.63,1.86],[0.0906278,-0.623397,0.71293,0.308049],[1,0,0,1],[9E+09,9E+09,9E+09,9E+09,9E+09,9E+09]], v20, seam13, weld13\Weave:=weave1, fine, tWeldGun;
		SingArea\Wrist;
		MoveL [[-158.90,1535.32,931.69],[0.0906389,-0.623348,0.712932,0.308139],[1,-2,1,0],[9E+09,9E+09,9E+09,9E+09,9E+09,9E+09]], vmax, z0, tWeldGun;
		MoveJ [[-173.66,614.72,251.09],[0.128906,0.0495871,0.95885,-0.248055],[1,-1,1,0],[9E+09,9E+09,9E+09,9E+09,9E+09,9E+09]], vmax, z0, tWeldGun;
		MoveL [[-145.55,555.68,15.34],[0.152232,0.0392509,0.96562,-0.207034],[1,-1,1,0],[9E+09,9E+09,9E+09,9E+09,9E+09,9E+09]], vmax, z0, tWeldGun;
		ArcLStart [[-145.25,553.61,5.23],[0.150684,0.0446148,0.957996,-0.239891],[1,-1,1,0],[9E+09,9E+09,9E+09,9E+09,9E+09,9E+09]], v20, seam13, weld13\Weave:=weave1, fine, tWeldGun;
		ArcLEnd [[-113.04,553.61,5.21],[0.150682,0.0446047,0.957994,-0.239902],[1,-1,1,0],[9E+09,9E+09,9E+09,9E+09,9E+09,9E+09]], v20, seam13, weld13\Weave:=weave1, fine, tWeldGun;
		MoveL [[-113.65,555.41,12.33],[0.152159,0.0393397,0.96563,-0.207027],[1,-1,1,0],[9E+09,9E+09,9E+09,9E+09,9E+09,9E+09]], vmax, z0, tWeldGun;
		MoveL [[173.88,557.63,12.23],[0.150918,0.0436625,0.959445,-0.234057],[1,-1,1,0],[9E+09,9E+09,9E+09,9E+09,9E+09,9E+09]], vmax, z0, tWeldGun;
		ArcLStart [[173.75,552.63,2.66],[0.150938,0.0436659,0.959441,-0.234061],[1,-1,1,0],[9E+09,9E+09,9E+09,9E+09,9E+09,9E+09]], v20, seam13, weld13\Weave:=weave1, fine, tWeldGun;
		ArcLEnd [[207.36,552.81,2.26],[0.150944,0.0436531,0.959435,-0.234083],[1,-1,1,0],[9E+09,9E+09,9E+09,9E+09,9E+09,9E+09]], v20, seam13, weld13\Weave:=weave1, fine, tWeldGun;
		MoveL [[207.49,559.40,13.87],[0.152119,0.0394488,0.965633,-0.20702],[1,-1,1,0],[9E+09,9E+09,9E+09,9E+09,9E+09,9E+09]], vmax, z0, tWeldGun;
		MoveL [[862.60,554.49,14.86],[0.152154,0.0392658,0.965627,-0.207055],[0,-2,1,0],[9E+09,9E+09,9E+09,9E+09,9E+09,9E+09]], vmax, z0, tWeldGun;
		ArcLStart [[864.91,549.07,1.34],[0.133495,0.0503347,0.954435,-0.262108],[0,-1,1,0],[9E+09,9E+09,9E+09,9E+09,9E+09,9E+09]], v20, seam13, weld13\Weave:=weave1, fine, tWeldGun;
		ArcLEnd [[899.31,549.07,1.33],[0.133493,0.0503325,0.954436,-0.262103],[0,-2,1,0],[9E+09,9E+09,9E+09,9E+09,9E+09,9E+09]], v20, seam13, weld13\Weave:=weave1, fine, tWeldGun;
		MoveL [[899.33,555.62,9.82],[0.152106,0.0393027,0.965639,-0.207029],[0,-2,1,0],[9E+09,9E+09,9E+09,9E+09,9E+09,9E+09]], vmax, z0, tWeldGun;
		MoveL [[1178.47,554.50,11.88],[0.149638,0.047924,0.952344,-0.261443],[0,-2,1,0],[9E+09,9E+09,9E+09,9E+09,9E+09,9E+09]], vmax, z0, tWeldGun;
		ArcLStart [[1182.61,548.27,-0.41],[0.119114,0.0614783,0.947533,-0.290197],[0,-2,1,0],[9E+09,9E+09,9E+09,9E+09,9E+09,9E+09]], v20, seam13, weld13\Weave:=weave1, fine, tWeldGun;
		ArcLEnd [[1211.37,548.80,-1.22],[0.119109,0.0614608,0.947531,-0.290208],[0,-2,1,0],[9E+09,9E+09,9E+09,9E+09,9E+09,9E+09]], v20, seam13, weld13\Weave:=weave1, fine, tWeldGun;
		MoveL [[1185.29,583.76,320.77],[0.152081,0.0394165,0.965666,-0.206898],[0,-2,1,0],[9E+09,9E+09,9E+09,9E+09,9E+09,9E+09]], vmax, z0, tWeldGun;
		MoveJ [[759.22,820.77,477.02],[0.128857,0.0495447,0.958803,-0.24827],[0,-1,1,0],[9E+09,9E+09,9E+09,9E+09,9E+09,9E+09]], vmax, z0, tWeldGun;
		MoveJ [[-401.88,982.38,420.80],[0.377905,-0.177501,-0.908663,-0.00353082],[1,0,1,0],[9E+09,9E+09,9E+09,9E+09,9E+09,9E+09]], vmax, z0, tWeldGun;
		MoveL [[-401.87,982.37,-5.96],[0.377901,-0.177501,-0.908665,-0.00352363],[1,0,1,0],[9E+09,9E+09,9E+09,9E+09,9E+09,9E+09]], v1000, z0, tWeldGun;
		ArcLStart [[-404.58,981.09,-7.78],[0.37795,-0.177396,-0.908665,-0.00362024],[1,0,1,0],[9E+09,9E+09,9E+09,9E+09,9E+09,9E+09]], v10, seam13, weld13\Weave:=weave1, fine, tWeldGun;
		ArcL [[-403.34,957.35,-6.28],[0.377997,-0.177583,-0.90861,-0.00339797],[1,0,1,0],[9E+09,9E+09,9E+09,9E+09,9E+09,9E+09]], v10, seam13, weld13\Weave:=weave1, z10, tWeldGun;
		ArcLEnd [[-425.46,950.14,-7.20],[0.197405,-0.679804,-0.668803,-0.227157],[1,0,2,0],[9E+09,9E+09,9E+09,9E+09,9E+09,9E+09]], v10, seam13, weld13\Weave:=weave1, fine, tWeldGun;
		MoveL [[-425.48,941.74,3.95],[0.197405,-0.679809,-0.668795,-0.227167],[1,0,2,0],[9E+09,9E+09,9E+09,9E+09,9E+09,9E+09]], vmax, z0, tWeldGun;
		MoveL [[-432.39,895.03,94.24],[0.274951,-0.581467,-0.743558,-0.182811],[1,0,2,0],[9E+09,9E+09,9E+09,9E+09,9E+09,9E+09]], vmax, z0, tWeldGun;
		MoveL [[-1101.20,895.02,94.24],[0.274939,-0.581469,-0.743563,-0.182805],[1,0,2,0],[9E+09,9E+09,9E+09,9E+09,9E+09,9E+09]], vmax, z0, tWeldGun;
		MoveL [[-1101.70,938.01,-1.40],[0.240452,-0.654006,-0.686015,-0.209388],[1,0,2,0],[9E+09,9E+09,9E+09,9E+09,9E+09,9E+09]], v1000, z0, tWeldGun;
		ArcLStart [[-1102.46,946.94,-5.88],[0.240345,-0.654194,-0.685887,-0.20934],[1,0,2,0],[9E+09,9E+09,9E+09,9E+09,9E+09,9E+09]], v10, seam13, weld13\Weave:=weave1, fine, tWeldGun;
		ArcL [[-1122.33,944.31,-5.63],[0.240415,-0.654059,-0.68597,-0.209414],[1,0,2,0],[9E+09,9E+09,9E+09,9E+09,9E+09,9E+09]], v10, seam13, weld13\Weave:=weave1, z10, tWeldGun;
		ArcLEnd [[-1131.87,975.46,-7.21],[0.0370294,0.922956,0.0834677,0.373919],[1,0,3,0],[9E+09,9E+09,9E+09,9E+09,9E+09,9E+09]], v10, seam13, weld13\Weave:=weave1, fine, tWeldGun;
		MoveL [[-1142.99,977.01,6.44],[0.0501214,0.923455,0.0523108,0.376805],[1,0,3,0],[9E+09,9E+09,9E+09,9E+09,9E+09,9E+09]], vmax, z0, tWeldGun;
		MoveJ [[-1224.84,979.29,303.50],[0.0444685,0.923113,0.0666376,0.376092],[1,0,-1,0],[9E+09,9E+09,9E+09,9E+09,9E+09,9E+09]], vmax, z20, tWeldGun;
		MoveL [[-1198.60,1154.71,4.46],[0.0444461,0.923123,0.0666424,0.37607],[1,0,-1,0],[9E+09,9E+09,9E+09,9E+09,9E+09,9E+09]], v1000, z0, tWeldGun;
		ArcLStart [[-1194.72,1155.51,-5.01],[0.0443844,0.92315,0.066588,0.376019],[1,0,-1,0],[9E+09,9E+09,9E+09,9E+09,9E+09,9E+09]], v10, seam13, weld13\Weave:=weave1, fine, tWeldGun;
		ArcL [[-1195.43,1176.10,-5.24],[0.044462,0.923146,0.0665592,0.376025],[1,0,-1,0],[9E+09,9E+09,9E+09,9E+09,9E+09,9E+09]], v10, seam13, weld13\Weave:=weave1, z10, tWeldGun;
		ArcLEnd [[-1167.22,1193.43,-4.61],[0.211529,0.696313,-0.654269,0.205758],[1,-1,0,0],[9E+09,9E+09,9E+09,9E+09,9E+09,9E+09]], v10, seam13, weld13\Weave:=weave1, fine, tWeldGun;
		MoveL [[-1165.81,1197.81,-4.44],[0.289046,0.665942,-0.622199,0.292988],[1,0,0,0],[9E+09,9E+09,9E+09,9E+09,9E+09,9E+09]], vmax, z0, tWeldGun;
		MoveL [[-1167.37,1197.80,267.48],[0.269054,0.631082,-0.684208,0.247398],[1,-1,0,0],[9E+09,9E+09,9E+09,9E+09,9E+09,9E+09]], vmax, z0, tWeldGun;
		MoveJ [[-491.85,1197.38,267.48],[0.269045,0.631086,-0.684208,0.247399],[1,-1,0,0],[9E+09,9E+09,9E+09,9E+09,9E+09,9E+09]], vmax, z0, tWeldGun;
		MoveL [[-493.75,1206.46,4.64],[0.230361,0.671978,-0.666396,0.226485],[1,-1,0,0],[9E+09,9E+09,9E+09,9E+09,9E+09,9E+09]], v1000, z0, tWeldGun;
		ArcLStart [[-496.53,1197.25,-8.21],[0.230282,0.672061,-0.666354,0.226445],[1,-1,0,0],[9E+09,9E+09,9E+09,9E+09,9E+09,9E+09]], v10, seam13, weld13\Weave:=weave1, fine, tWeldGun;
		ArcL [[-474.00,1197.10,-7.28],[0.230378,0.67197,-0.666403,0.226474],[1,-1,0,0],[9E+09,9E+09,9E+09,9E+09,9E+09,9E+09]], v10, seam13, weld13\Weave:=weave1, z10, tWeldGun;
		ArcLEnd [[-464.66,1164.90,-10.34],[0.384973,0.00807935,-0.922617,-0.0225858],[1,-1,1,0],[9E+09,9E+09,9E+09,9E+09,9E+09,9E+09]], v10, seam13, weld13\Weave:=weave1, fine, tWeldGun;
		MoveL [[-460.21,1166.10,-6.29],[0.384934,0.00803439,-0.922633,-0.0226006],[1,-1,1,0],[9E+09,9E+09,9E+09,9E+09,9E+09,9E+09]], vmax, z5, tWeldGun;
		MoveL [[-460.61,1166.13,158.38],[0.384913,0.00804793,-0.922641,-0.0226089],[1,-1,1,0],[9E+09,9E+09,9E+09,9E+09,9E+09,9E+09]], vmax, z5, tWeldGun;
		MoveJ [[-411.67,714.00,66.77],[0.262804,0.646065,-0.670013,0.254199],[1,-1,0,0],[9E+09,9E+09,9E+09,9E+09,9E+09,9E+09]], vmax, z5, tWeldGun;
		MoveL [[-412.17,719.36,-3.08],[0.242994,0.661127,-0.665052,0.248138],[1,-1,0,0],[9E+09,9E+09,9E+09,9E+09,9E+09,9E+09]], vmax, z5, tWeldGun;
		ArcLStart [[-411.29,716.55,-6.44],[0.220122,0.668768,-0.676858,0.214847],[1,-1,0,0],[9E+09,9E+09,9E+09,9E+09,9E+09,9E+09]], v5, seam13, weld13\Weave:=weave1, fine, tWeldGun;
		ArcLEnd [[-430.47,716.55,-6.45],[0.220123,0.668765,-0.676857,0.214859],[1,-1,0,0],[9E+09,9E+09,9E+09,9E+09,9E+09,9E+09]], v5, seam13, weld13\Weave:=weave1, fine, tWeldGun;
		MoveL [[-433.52,712.50,86.63],[0.256209,0.656106,-0.660016,0.261269],[1,-1,0,0],[9E+09,9E+09,9E+09,9E+09,9E+09,9E+09]], vmax, z5, tWeldGun;
		MoveL [[-1103.37,713.70,123.92],[0.256219,0.656103,-0.660014,0.261271],[1,-1,0,0],[9E+09,9E+09,9E+09,9E+09,9E+09,9E+09]], vmax, z5, tWeldGun;
		MoveL [[-1103.35,717.29,-4.25],[0.256222,0.656097,-0.66001,0.261295],[1,-1,0,0],[9E+09,9E+09,9E+09,9E+09,9E+09,9E+09]], vmax, z5, tWeldGun;
		ArcLStart [[-1103.12,713.69,-5.87],[0.256215,0.656125,-0.659976,0.261315],[1,-1,0,0],[9E+09,9E+09,9E+09,9E+09,9E+09,9E+09]], v5, seam13, weld13\Weave:=weave1, fine, tWeldGun;
		ArcLEnd [[-1123.49,713.72,-5.89],[0.256214,0.656129,-0.659971,0.26132],[1,-1,0,0],[9E+09,9E+09,9E+09,9E+09,9E+09,9E+09]], v5, seam13, weld13\Weave:=weave1, fine, tWeldGun;
		MoveL [[-1124.57,723.78,145.38],[0.256225,0.656093,-0.660015,0.261287],[1,-1,0,0],[9E+09,9E+09,9E+09,9E+09,9E+09,9E+09]], vmax, z5, tWeldGun;
		MoveJ [[-1174.22,1417.20,153.64],[0.288404,-0.63354,-0.657568,-0.288193],[1,-1,-2,0],[9E+09,9E+09,9E+09,9E+09,9E+09,9E+09]], vmax, z5, tWeldGun;
		MoveL [[-1185.47,1420.19,5.39],[0.288267,-0.633625,-0.657572,-0.288135],[1,-1,-2,0],[9E+09,9E+09,9E+09,9E+09,9E+09,9E+09]], vmax, z5, tWeldGun;
		ArcLStart [[-1185.37,1426.63,-5.37],[0.288326,-0.633566,-0.657577,-0.288195],[1,-1,-2,0],[9E+09,9E+09,9E+09,9E+09,9E+09,9E+09]], v5, seam13, weld13\Weave:=weave1, fine, tWeldGun;
		ArcLEnd [[-1164.37,1426.62,-5.55],[0.288311,-0.633564,-0.657587,-0.28819],[1,-1,-2,0],[9E+09,9E+09,9E+09,9E+09,9E+09,9E+09]], v5, seam13, weld13\Weave:=weave1, fine, tWeldGun;
		MoveL [[-1165.69,1421.27,86.72],[0.28839,-0.633573,-0.657541,-0.288197],[1,-1,-2,0],[9E+09,9E+09,9E+09,9E+09,9E+09,9E+09]], vmax, z5, tWeldGun;
		MoveL [[-494.06,1426.01,134.66],[0.280642,-0.634844,-0.656104,-0.296212],[1,-1,-2,0],[9E+09,9E+09,9E+09,9E+09,9E+09,9E+09]], vmax, z5, tWeldGun;
		MoveL [[-492.29,1423.04,-11.79],[0.251513,-0.647275,-0.667795,-0.268004],[1,-1,-2,0],[9E+09,9E+09,9E+09,9E+09,9E+09,9E+09]], vmax, z5, tWeldGun;
		ArcLStart [[-491.87,1429.46,-11.99],[0.251491,-0.647295,-0.667791,-0.267988],[1,-1,-2,0],[9E+09,9E+09,9E+09,9E+09,9E+09,9E+09]], v5, seam13, weld13\Weave:=weave1, fine, tWeldGun;
		ArcLEnd [[-472.07,1429.61,-12.01],[0.251461,-0.647305,-0.667793,-0.267986],[1,-1,-2,0],[9E+09,9E+09,9E+09,9E+09,9E+09,9E+09]], v5, seam13, weld13\Weave:=weave1, fine, tWeldGun;
		MoveL [[-471.84,1418.41,452.48],[0.280608,-0.634847,-0.656147,-0.296143],[1,-1,-2,0],[9E+09,9E+09,9E+09,9E+09,9E+09,9E+09]], vmax, z5, tWeldGun;
		MoveJ pSafeS1, vmax, fine, tWeldGun;
	ENDPROC
	PROC ss_200()
           	rTestPosTop;
		TPWrite "Side 1 A";
		MoveJ pSafeS1, vmax, fine, tWeldGun;
		!Code Goes Here
		MoveJ pSafeS181, vmax, fine, tWeldGun;
		SingArea\Wrist;
		MoveJ [[1181.97,1536.60,299.24],[0.0635588,0.517232,-0.779106,0.348462],[0,1,-3,1],[9E+09,9E+09,9E+09,9E+09,9E+09,9E+09]], vmax, z10, tWeldGun;
		MoveL [[1181.96,1536.60,-12.62],[0.0635661,0.517237,-0.779104,0.348458],[0,1,-2,1],[9E+09,9E+09,9E+09,9E+09,9E+09,9E+09]], v1000, z10, tWeldGun;
		ArcLStart [[1181.53,1529.02,-11.65],[0.0635714,0.517237,-0.779104,0.348457],[0,1,-2,1],[9E+09,9E+09,9E+09,9E+09,9E+09,9E+09]], v10, seam13, weld13\Weave:=weave1, fine, tWeldGun;
		ArcLEnd [[1204.96,1529.87,-10.62],[0.0635614,0.517237,-0.779103,0.348461],[0,1,-2,1],[9E+09,9E+09,9E+09,9E+09,9E+09,9E+09]], v10, seam13, weld13\Weave:=weave1, fine, tWeldGun;
		MoveL [[1204.64,1537.23,-12.62],[0.0635617,0.517239,-0.7791,0.348464],[0,1,-2,1],[9E+09,9E+09,9E+09,9E+09,9E+09,9E+09]], vmax, z10, tWeldGun;
		MoveL [[863.66,1538.85,77.89],[0.0635666,0.517243,-0.779097,0.348464],[0,1,-2,1],[9E+09,9E+09,9E+09,9E+09,9E+09,9E+09]], vmax, z10, tWeldGun;
		MoveJ [[861.58,1461.21,260.09],[0.14949,-0.376148,-0.839997,-0.361347],[0,1,-1,1],[9E+09,9E+09,9E+09,9E+09,9E+09,9E+09]], vmax, z10, tWeldGun;
		MoveL [[863.23,1471.68,-11.89],[0.149517,-0.37621,-0.839967,-0.361342],[0,1,-1,1],[9E+09,9E+09,9E+09,9E+09,9E+09,9E+09]], v1000, z10, tWeldGun;
		ArcLStart [[863.88,1474.96,-12.64],[0.149558,-0.376296,-0.839897,-0.361396],[0,1,-1,1],[9E+09,9E+09,9E+09,9E+09,9E+09,9E+09]], v10, seam13, weld13\Weave:=weave1, fine, tWeldGun;
		ArcLEnd [[887.67,1475.21,-13.25],[0.149548,-0.376266,-0.839942,-0.361327],[0,1,-1,1],[9E+09,9E+09,9E+09,9E+09,9E+09,9E+09]], v10, seam13, weld13\Weave:=weave1, fine, tWeldGun;
		MoveL [[886.08,1463.03,-7.28],[0.149478,-0.376156,-0.840008,-0.361317],[0,1,-1,1],[9E+09,9E+09,9E+09,9E+09,9E+09,9E+09]], vmax, z10, tWeldGun;
		MoveJ [[863.35,1506.96,224.59],[0.0635605,0.517248,-0.779091,0.348471],[0,1,-2,1],[9E+09,9E+09,9E+09,9E+09,9E+09,9E+09]], vmax, z10, tWeldGun;
		MoveL [[863.21,1535.55,-10.64],[0.0635626,0.51725,-0.779093,0.348463],[0,1,-2,1],[9E+09,9E+09,9E+09,9E+09,9E+09,9E+09]], vmax, z10, tWeldGun;
		ArcLStart [[862.98,1531.20,-11.14],[0.0635851,0.517245,-0.779094,0.348464],[0,1,-2,1],[9E+09,9E+09,9E+09,9E+09,9E+09,9E+09]], v10, seam13, weld13\Weave:=weave1, fine, tWeldGun;
		ArcLEnd [[887.38,1530.81,-10.94],[0.0635922,0.517251,-0.779089,0.348465],[0,1,-2,1],[9E+09,9E+09,9E+09,9E+09,9E+09,9E+09]], v10, seam13, weld13\Weave:=weave1, fine, tWeldGun;
		MoveL [[887.77,1539.90,182.89],[0.0635615,0.517251,-0.779088,0.348474],[0,1,-2,1],[9E+09,9E+09,9E+09,9E+09,9E+09,9E+09]], vmax, z10, tWeldGun;
		MoveJ [[1182.52,1470.34,61.27],[0.149538,-0.376243,-0.839941,-0.361358],[0,1,-1,1],[9E+09,9E+09,9E+09,9E+09,9E+09,9E+09]], vmax, z10, tWeldGun;
		MoveL [[1182.53,1470.34,-16.07],[0.149529,-0.376231,-0.83995,-0.361353],[0,1,-1,1],[9E+09,9E+09,9E+09,9E+09,9E+09,9E+09]], v1000, z10, tWeldGun;
		ArcLStart [[1181.99,1475.51,-15.52],[0.149552,-0.376279,-0.83992,-0.361363],[0,1,-1,1],[9E+09,9E+09,9E+09,9E+09,9E+09,9E+09]], v10, seam13, weld13\Weave:=weave1, fine, tWeldGun;
		ArcLEnd [[1204.38,1476.47,-15.60],[0.149569,-0.376356,-0.839878,-0.361375],[0,1,-1,1],[9E+09,9E+09,9E+09,9E+09,9E+09,9E+09]], v10, seam13, weld13\Weave:=weave1, fine, tWeldGun;
		MoveL [[1202.33,1469.98,-15.09],[0.149549,-0.376274,-0.839922,-0.361365],[0,1,-1,1],[9E+09,9E+09,9E+09,9E+09,9E+09,9E+09]], vmax, z10, tWeldGun;
		MoveL [[1203.94,921.98,77.52],[0.149416,-0.376356,-0.839957,-0.361252],[0,1,-1,1],[9E+09,9E+09,9E+09,9E+09,9E+09,9E+09]], vmax, z10, tWeldGun;
		MoveL [[1203.94,921.99,-12.97],[0.149422,-0.376348,-0.839957,-0.361259],[0,1,-1,1],[9E+09,9E+09,9E+09,9E+09,9E+09,9E+09]], v1000, z10, tWeldGun;
		ArcLStart [[1203.94,928.79,-14.21],[0.149423,-0.376362,-0.839952,-0.361256],[0,1,-1,1],[9E+09,9E+09,9E+09,9E+09,9E+09,9E+09]], v10, seam13, weld13\Weave:=weave1, fine, tWeldGun;
		ArcLEnd [[1178.19,928.79,-14.21],[0.149422,-0.376442,-0.839904,-0.361285],[0,1,-1,1],[9E+09,9E+09,9E+09,9E+09,9E+09,9E+09]], v10, seam13, weld13\Weave:=weave1, fine, tWeldGun;
		MoveL [[1177.78,921.50,-1.65],[0.149422,-0.376364,-0.839949,-0.36126],[0,1,-1,1],[9E+09,9E+09,9E+09,9E+09,9E+09,9E+09]], vmax, z10, tWeldGun;
		MoveL [[883.71,921.14,-1.64],[0.149424,-0.37639,-0.839933,-0.361269],[0,1,0,1],[9E+09,9E+09,9E+09,9E+09,9E+09,9E+09]], vmax, z10, tWeldGun;
		MoveL [[883.71,926.93,-12.24],[0.149423,-0.3764,-0.839927,-0.361273],[0,0,0,1],[9E+09,9E+09,9E+09,9E+09,9E+09,9E+09]], v1000, z10, tWeldGun;
		ArcLStart [[885.40,928.75,-13.38],[0.149454,-0.376503,-0.839867,-0.361295],[0,0,0,1],[9E+09,9E+09,9E+09,9E+09,9E+09,9E+09]], v10, seam13, weld13\Weave:=weave1, fine, tWeldGun;
		ArcLEnd [[866.41,928.73,-13.39],[0.149444,-0.376494,-0.839881,-0.361275],[0,0,0,1],[9E+09,9E+09,9E+09,9E+09,9E+09,9E+09]], v10, seam13, weld13\Weave:=weave1, fine, tWeldGun;
		MoveL [[863.70,926.54,-12.25],[0.149435,-0.37642,-0.839913,-0.361282],[0,0,0,1],[9E+09,9E+09,9E+09,9E+09,9E+09,9E+09]], v100, z10, tWeldGun;
		MoveL [[861.26,919.79,117.88],[0.149443,-0.376442,-0.8399,-0.361285],[0,1,-1,1],[9E+09,9E+09,9E+09,9E+09,9E+09,9E+09]], vmax, z0, tWeldGun;
		MoveJ [[868.17,991.07,127.71],[0.0426372,-0.330552,0.858067,-0.39069],[0,1,-2,1],[9E+09,9E+09,9E+09,9E+09,9E+09,9E+09]], vmax, z0, tWeldGun;
		MoveL [[868.52,991.54,-9.45],[0.0429862,-0.330642,0.857997,-0.390729],[0,0,-2,1],[9E+09,9E+09,9E+09,9E+09,9E+09,9E+09]], v1000, z10, tWeldGun;
		ArcLStart [[865.93,978.35,-10.52],[0.0429801,-0.330651,0.857991,-0.390736],[0,0,-2,1],[9E+09,9E+09,9E+09,9E+09,9E+09,9E+09]], v10, seam13, weld13\Weave:=weave1, fine, tWeldGun;
		ArcLEnd [[888.37,978.36,-11.00],[0.0429914,-0.330695,0.857973,-0.390738],[0,0,-2,1],[9E+09,9E+09,9E+09,9E+09,9E+09,9E+09]], v10, seam13, weld13\Weave:=weave1, fine, tWeldGun;
		MoveL [[889.59,992.71,-9.41],[0.0430222,-0.330607,0.858002,-0.390746],[0,0,-2,1],[9E+09,9E+09,9E+09,9E+09,9E+09,9E+09]], vmax, z10, tWeldGun;
		MoveL [[889.59,992.73,75.52],[0.0430306,-0.330621,0.857997,-0.390743],[0,1,-2,1],[9E+09,9E+09,9E+09,9E+09,9E+09,9E+09]], vmax, z10, tWeldGun;
		MoveL [[1177.66,992.72,75.52],[0.0430182,-0.33062,0.857997,-0.390745],[0,0,-2,1],[9E+09,9E+09,9E+09,9E+09,9E+09,9E+09]], vmax, z10, tWeldGun;
		MoveL [[1185.41,992.70,-11.53],[0.0429716,-0.330606,0.858007,-0.390739],[0,0,-2,1],[9E+09,9E+09,9E+09,9E+09,9E+09,9E+09]], v1000, z10, tWeldGun;
		ArcLStart [[1180.66,978.10,-13.63],[0.0429557,-0.330625,0.857997,-0.390747],[0,0,-2,1],[9E+09,9E+09,9E+09,9E+09,9E+09,9E+09]], v10, seam13, weld13\Weave:=weave1, fine, tWeldGun;
		ArcLEnd [[1207.05,977.71,-13.62],[0.0429527,-0.330628,0.857994,-0.390751],[0,0,-2,1],[9E+09,9E+09,9E+09,9E+09,9E+09,9E+09]], v10, seam13, weld13\Weave:=weave1, fine, tWeldGun;
		MoveL [[1207.94,989.04,-11.16],[0.0429397,-0.330625,0.858002,-0.39074],[0,0,-2,1],[9E+09,9E+09,9E+09,9E+09,9E+09,9E+09]], v1000, z10, tWeldGun;
		MoveL [[1207.95,989.04,392.36],[0.0429563,-0.330627,0.857995,-0.39075],[0,1,-2,1],[9E+09,9E+09,9E+09,9E+09,9E+09,9E+09]], vmax, z10, tWeldGun;
		MoveJ [[194.09,1536.38,108.42],[0.0907205,-0.623393,0.712906,0.308084],[0,-1,0,1],[9E+09,9E+09,9E+09,9E+09,9E+09,9E+09]], vmax, z10, tWeldGun;
		MoveL [[194.09,1534.55,44.51],[0.0907126,-0.623398,0.712901,0.308089],[0,-1,0,1],[9E+09,9E+09,9E+09,9E+09,9E+09,9E+09]], vmax, z10, tWeldGun;
		ArcLStart [[191.25,1532.54,0.05],[0.0904838,-0.623408,0.712969,0.30798],[0,-1,0,1],[9E+09,9E+09,9E+09,9E+09,9E+09,9E+09]], v20, seam13, weld13\Weave:=weave1, fine, tWeldGun;
		ArcLEnd [[157.22,1532.54,0.51],[0.090482,-0.623409,0.712967,0.307981],[0,-1,0,1],[9E+09,9E+09,9E+09,9E+09,9E+09,9E+09]], v20, seam13, weld13\Weave:=weave1, fine, tWeldGun;
		MoveL [[158.09,1532.35,8.43],[0.0907075,-0.623402,0.712898,0.30809],[0,-1,0,1],[9E+09,9E+09,9E+09,9E+09,9E+09,9E+09]], vmax, z10, tWeldGun;
		MoveL [[-123.91,1535.35,12.43],[0.0907124,-0.623396,0.712903,0.308089],[1,0,0,1],[9E+09,9E+09,9E+09,9E+09,9E+09,9E+09]], vmax, z10, tWeldGun;
		ArcLStart [[-126.92,1534.33,1.43],[0.0907044,-0.623405,0.712895,0.308091],[1,0,0,1],[9E+09,9E+09,9E+09,9E+09,9E+09,9E+09]], v20, seam13, weld13\Weave:=weave1, fine, tWeldGun;
		ArcLEnd [[-160.92,1534.33,1.44],[0.090708,-0.623403,0.712896,0.308092],[1,0,0,1],[9E+09,9E+09,9E+09,9E+09,9E+09,9E+09]], v20, seam13, weld13\Weave:=weave1, fine, tWeldGun;
		MoveL [[-158.90,1535.32,931.69],[0.0906389,-0.623348,0.712932,0.308139],[1,-2,1,0],[9E+09,9E+09,9E+09,9E+09,9E+09,9E+09]], vmax, z0, tWeldGun;
		MoveJ [[-173.66,614.72,251.09],[0.128906,0.0495871,0.95885,-0.248055],[1,-1,1,0],[9E+09,9E+09,9E+09,9E+09,9E+09,9E+09]], vmax, z0, tWeldGun;
		MoveL [[-146.66,553.40,15.33],[0.15216,0.0393582,0.96563,-0.207021],[1,-1,1,0],[9E+09,9E+09,9E+09,9E+09,9E+09,9E+09]], vmax, z0, tWeldGun;
		ArcLStart [[-146.66,553.39,2.32],[0.152156,0.0393511,0.965628,-0.207036],[1,-1,1,0],[9E+09,9E+09,9E+09,9E+09,9E+09,9E+09]], v20, seam13, weld13\Weave:=weave1, fine, tWeldGun;
		ArcLEnd [[-114.67,554.39,1.31],[0.152148,0.0393507,0.965628,-0.207043],[1,-1,1,0],[9E+09,9E+09,9E+09,9E+09,9E+09,9E+09]], v20, seam13, weld13\Weave:=weave1, fine, tWeldGun;
		MoveL [[-113.65,555.41,12.33],[0.152159,0.0393397,0.96563,-0.207027],[1,-1,1,0],[9E+09,9E+09,9E+09,9E+09,9E+09,9E+09]], vmax, z0, tWeldGun;
		MoveL [[171.61,552.68,21.42],[0.152083,0.0394694,0.965633,-0.207041],[1,-1,1,0],[9E+09,9E+09,9E+09,9E+09,9E+09,9E+09]], vmax, z0, tWeldGun;
		ArcLStart [[171.63,552.69,-0.51],[0.152132,0.0394445,0.96562,-0.207073],[1,-1,1,0],[9E+09,9E+09,9E+09,9E+09,9E+09,9E+09]], v20, seam13, weld13\Weave:=weave1, fine, tWeldGun;
		ArcLEnd [[202.63,552.69,-0.52],[0.152129,0.0394303,0.965618,-0.207083],[1,-1,1,0],[9E+09,9E+09,9E+09,9E+09,9E+09,9E+09]], v20, seam13, weld13\Weave:=weave1, fine, tWeldGun;
		MoveL [[204.25,552.75,13.91],[0.152145,0.0394344,0.965619,-0.207068],[1,-1,1,0],[9E+09,9E+09,9E+09,9E+09,9E+09,9E+09]], vmax, z0, tWeldGun;
		MoveL [[860.18,549.11,14.83],[0.152112,0.039289,0.965636,-0.207043],[0,-2,1,0],[9E+09,9E+09,9E+09,9E+09,9E+09,9E+09]], vmax, z0, tWeldGun;
		ArcLStart [[860.21,550.17,-4.16],[0.152159,0.0392088,0.965632,-0.207039],[0,-2,1,0],[9E+09,9E+09,9E+09,9E+09,9E+09,9E+09]], v20, seam13, weld13\Weave:=weave1, fine, tWeldGun;
		ArcLEnd [[895.96,549.20,-3.18],[0.152141,0.039174,0.965634,-0.207051],[0,-2,1,0],[9E+09,9E+09,9E+09,9E+09,9E+09,9E+09]], v20, seam13, weld13\Weave:=weave1, fine, tWeldGun;
		MoveL [[895.37,549.34,9.83],[0.15211,0.0392827,0.965635,-0.207047],[0,-2,1,0],[9E+09,9E+09,9E+09,9E+09,9E+09,9E+09]], vmax, z0, tWeldGun;
		MoveL [[1175.32,546.94,11.83],[0.1496,0.0478929,0.95235,-0.261449],[0,-2,1,0],[9E+09,9E+09,9E+09,9E+09,9E+09,9E+09]], vmax, z0, tWeldGun;
		ArcLStart [[1177.31,546.94,-3.16],[0.149595,0.0478934,0.95235,-0.261454],[0,-2,1,0],[9E+09,9E+09,9E+09,9E+09,9E+09,9E+09]], v20, seam13, weld13\Weave:=weave1, fine, tWeldGun;
		ArcLEnd [[1209.31,546.95,-3.16],[0.149595,0.0478909,0.95235,-0.261454],[0,-2,1,0],[9E+09,9E+09,9E+09,9E+09,9E+09,9E+09]], v20, seam13, weld13\Weave:=weave1, fine, tWeldGun;
		MoveL [[1183.76,537.75,320.86],[0.152128,0.0394118,0.965637,-0.207003],[0,-2,1,0],[9E+09,9E+09,9E+09,9E+09,9E+09,9E+09]], vmax, z0, tWeldGun;
		MoveJ [[759.22,820.77,477.02],[0.128857,0.0495447,0.958803,-0.24827],[0,-1,1,0],[9E+09,9E+09,9E+09,9E+09,9E+09,9E+09]], vmax, z0, tWeldGun;
		MoveJ [[-401.88,982.38,420.80],[0.377905,-0.177501,-0.908663,-0.00353082],[1,0,1,0],[9E+09,9E+09,9E+09,9E+09,9E+09,9E+09]], vmax, z0, tWeldGun;
		MoveL [[-401.87,982.37,-5.96],[0.377901,-0.177501,-0.908665,-0.00352363],[1,0,1,0],[9E+09,9E+09,9E+09,9E+09,9E+09,9E+09]], v1000, z0, tWeldGun;
		ArcLStart [[-407.18,982.54,-5.95],[0.377941,-0.177364,-0.908675,-0.00361829],[1,0,1,0],[9E+09,9E+09,9E+09,9E+09,9E+09,9E+09]], v10, seam13, weld13\Weave:=weave1, fine, tWeldGun;
		ArcL [[-407.21,961.97,-7.34],[0.377917,-0.177516,-0.908656,-0.00352015],[1,0,1,0],[9E+09,9E+09,9E+09,9E+09,9E+09,9E+09]], v10, seam13, weld13\Weave:=weave1, z10, tWeldGun;
		ArcLEnd [[-429.48,955.83,-6.96],[0.274941,-0.581479,-0.743555,-0.1828],[1,0,2,0],[9E+09,9E+09,9E+09,9E+09,9E+09,9E+09]], v10, seam13, weld13\Weave:=weave1, fine, tWeldGun;
		MoveL [[-432.47,945.01,-6.78],[0.274937,-0.581449,-0.743579,-0.182803],[1,0,2,0],[9E+09,9E+09,9E+09,9E+09,9E+09,9E+09]], vmax, z0, tWeldGun;
		MoveL [[-432.39,895.03,94.24],[0.274951,-0.581467,-0.743558,-0.182811],[1,0,2,0],[9E+09,9E+09,9E+09,9E+09,9E+09,9E+09]], vmax, z0, tWeldGun;
		MoveL [[-1101.20,895.02,94.24],[0.274939,-0.581469,-0.743563,-0.182805],[1,0,2,0],[9E+09,9E+09,9E+09,9E+09,9E+09,9E+09]], vmax, z0, tWeldGun;
		MoveL [[-1101.21,942.37,-3.25],[0.274946,-0.581512,-0.743526,-0.182807],[1,0,2,0],[9E+09,9E+09,9E+09,9E+09,9E+09,9E+09]], v1000, z0, tWeldGun;
		ArcLStart [[-1099.81,952.01,-6.02],[0.23841,-0.593999,-0.734594,-0.225162],[1,0,2,0],[9E+09,9E+09,9E+09,9E+09,9E+09,9E+09]], v10, seam13, weld13\Weave:=weave1, fine, tWeldGun;
		ArcL [[-1121.08,951.80,-5.63],[0.238289,-0.634044,-0.696044,-0.238181],[1,0,2,0],[9E+09,9E+09,9E+09,9E+09,9E+09,9E+09]], v10, seam13, weld13\Weave:=weave1, z10, tWeldGun;
		ArcLEnd [[-1129.28,975.89,-6.00],[0.0369776,0.92297,0.0835389,0.373873],[1,0,3,0],[9E+09,9E+09,9E+09,9E+09,9E+09,9E+09]], v10, seam13, weld13\Weave:=weave1, fine, tWeldGun;
		MoveL [[-1142.99,977.01,6.44],[0.0501214,0.923455,0.0523108,0.376805],[1,0,3,0],[9E+09,9E+09,9E+09,9E+09,9E+09,9E+09]], vmax, z0, tWeldGun;
		MoveJ [[-1142.58,979.31,303.50],[0.0444513,0.923112,0.0666342,0.376096],[1,0,-1,0],[9E+09,9E+09,9E+09,9E+09,9E+09,9E+09]], vmax, z20, tWeldGun;
		MoveL [[-1192.76,1156.53,-4.42],[0.044443,0.923122,0.0666432,0.376072],[1,0,-1,0],[9E+09,9E+09,9E+09,9E+09,9E+09,9E+09]], v1000, z0, tWeldGun;
		ArcLStart [[-1192.23,1155.72,-3.63],[0.0444473,0.923132,0.0666323,0.376048],[1,0,-1,0],[9E+09,9E+09,9E+09,9E+09,9E+09,9E+09]], v10, seam13, weld13\Weave:=weave1, fine, tWeldGun;
		ArcL [[-1191.71,1175.69,-5.33],[0.0444379,0.923126,0.0666324,0.376065],[1,0,-1,0],[9E+09,9E+09,9E+09,9E+09,9E+09,9E+09]], v10, seam13, weld13\Weave:=weave1, z10, tWeldGun;
		ArcLEnd [[-1165.81,1187.00,-4.44],[0.28905,0.665936,-0.622204,0.292989],[1,0,0,0],[9E+09,9E+09,9E+09,9E+09,9E+09,9E+09]], v10, seam13, weld13\Weave:=weave1, fine, tWeldGun;
		MoveL [[-1165.81,1197.81,-4.44],[0.289046,0.665942,-0.622199,0.292988],[1,0,0,0],[9E+09,9E+09,9E+09,9E+09,9E+09,9E+09]], vmax, z0, tWeldGun;
		MoveL [[-1167.37,1197.80,267.48],[0.269054,0.631082,-0.684208,0.247398],[1,-1,0,0],[9E+09,9E+09,9E+09,9E+09,9E+09,9E+09]], vmax, z0, tWeldGun;
		MoveJ [[-491.85,1197.38,267.48],[0.269045,0.631086,-0.684208,0.247399],[1,-1,0,0],[9E+09,9E+09,9E+09,9E+09,9E+09,9E+09]], vmax, z0, tWeldGun;
		MoveL [[-495.49,1197.07,-6.30],[0.260132,0.661057,-0.654909,0.257739],[1,-1,0,0],[9E+09,9E+09,9E+09,9E+09,9E+09,9E+09]], v1000, z0, tWeldGun;
		ArcLStart [[-495.49,1192.07,-6.30],[0.260133,0.661061,-0.654906,0.257736],[1,-1,0,0],[9E+09,9E+09,9E+09,9E+09,9E+09,9E+09]], v10, seam13, weld13\Weave:=weave1, fine, tWeldGun;
		ArcL [[-474.53,1190.57,-6.48],[0.263861,0.655019,-0.660957,0.253897],[1,-1,0,0],[9E+09,9E+09,9E+09,9E+09,9E+09,9E+09]], v10, seam13, weld13\Weave:=weave1, z10, tWeldGun;
		ArcLEnd [[-467.21,1164.88,-8.10],[0.384925,0.00804232,-0.922637,-0.0225898],[1,-1,1,0],[9E+09,9E+09,9E+09,9E+09,9E+09,9E+09]], v10, seam13, weld13\Weave:=weave1, fine, tWeldGun;
		MoveL [[-460.21,1166.10,-6.29],[0.384934,0.00803439,-0.922633,-0.0226006],[1,-1,1,0],[9E+09,9E+09,9E+09,9E+09,9E+09,9E+09]], vmax, z5, tWeldGun;
		MoveL [[-460.61,1166.12,771.55],[0.384916,0.00803537,-0.92264,-0.0226078],[1,-1,1,0],[9E+09,9E+09,9E+09,9E+09,9E+09,9E+09]], vmax, z5, tWeldGun;
		MoveJ pSafeS1, vmax, fine, tWeldGun;
	ENDPROC

